VAR_GLOBAL CONSTANT
	cRECVDATACHANNELBUFFER: INT := 20;
END_VAR

(* stored: Version 1.1.0.1, ProductVersion 3.1.0.26
   GVL IdBaseConst: Id {3b5050a6-43fb-4c78-b1e7-56d2e896ad1a} *)
